FUNCTION_BLOCK FB_SaMElementWashing EXTENDS FB_SaMElement
VAR
END_VAR

END_FUNCTION_BLOCK

(* stored: Version 1.1.0.1
   POU FB_SaMElementWashing: Id {ef533864-744c-0365-03e8-3819c383dbae}, SpecialFunc None *)
